TYPE ST_SCANNER_Status :   //ST_SCANNER
STRUCT
	
	nState	: BYTE;
	
	I		: ST_SCANNER_IN;
	Q		: ST_SCANNER_OUT;
	
END_STRUCT
END_TYPE

(* stored: Version 1.1.0.1
   DUT ST_SCANNER_Status: Id {57af2c47-c610-4640-bc4a-ac973c87570b} *)
